/// calibration that is determined by calibration sequences of the unit (static offsets, shifts)
TYPE DrillingDataCalibration :
STRUCT
END_STRUCT
END_TYPE

(* stored: Version 1.1.0.1
   DUT DrillingDataCalibration: Id {b8e8fd06-4128-4bf9-bc97-b0e999aa021c} *)
